FUNCTION_BLOCK FB_Euchner_MBM
VAR_INPUT
	stHwIn: ST_Euchner_MBM_HW_IN;
	bReset: BOOL;
END_VAR
VAR_OUTPUT
	stHwOut: ST_Euchner_MBM_HW_OUT;
	bError: BOOL;
	stErrorText: ST_Text;
END_VAR
VAR
	stIn: ST_Euchner_MBM_IN;
	stOut: ST_Euchner_MBM_Out;
	tonReset: ton;
END_VAR

M_Mapping();
M_Supervision();

tonReset.IN := bReset;
tonReset.PT := T#150MS;
tonReset();
IF tonReset.Q THEN
	bReset := FALSE;
END_IF
stOut.bBM_ACK_G := bReset;

METHOD PRIVATE M_Error : BOOL
VAR_INPUT
	stError: ST_Text;
END_VAR
bError	:=TRUE;
stErrorText	:= stError;
END_METHOD

METHOD PRIVATE M_Mapping : BOOL
//mapping in
stIn.bBM_D_RUN := stHwIn.nByte0.0;
stIn.bBM_E_ML1 := stHwIn.nByte0.1;
stIn.bBM_E_ML2 := stHwIn.nByte0.2;
stIn.bBM_E_SYS := stHwIn.nByte0.3;
stIn.bBM_E_G := stHwIn.nByte0.4;

//mapping in
stHwOut.nByte0.0 := stOut.bBM_ACK_G;
END_METHOD

METHOD M_Reset : BOOL
bReset	:= TRUE;
bError	:= FALSE;
MEMSET(ADR(stErrorText), 0, SiZEOF(stErrorText));
END_METHOD

METHOD PRIVATE M_Supervision : BOOL
IF stIn.bBM_E_ML1 THEN
	M_Error(F_CreateDynTextDefault("Fehler Modul MBM Starng 1")); 	
ELSIF stIn.bBM_E_ML1 THEN
	M_Error(F_CreateDynTextDefault("Fehler Modul MBM Starng 1"));	
ELSIF stIn.bBM_E_G THEN
	M_Error(F_CreateDynTextDefault("Modul MBM Allgemein"));	
ELSIF stIn.bBM_E_SYS THEN
	M_Error(F_CreateDynTextDefault("Fehler Gesamtsystem"));
END_IF
END_METHOD

END_FUNCTION_BLOCK

(* stored: Version 1.1.0.1, ProductVersion 3.1.4024.12
   POU FB_Euchner_MBM: Id {454bc480-5abf-482e-879d-5005b27308c6}, SpecialFunc None
   Method M_Error: Id {f1921ebe-4704-4a35-a03a-8bf4df5b7517}
   Method M_Mapping: Id {d872bef3-b263-479d-a742-1009d3f3c85c}
   Method M_Reset: Id {8eaf9f2b-a058-4afe-8a85-01e309ea6655}
   Method M_Supervision: Id {a4000f4a-8800-48ba-a97d-98e4ecf8db56} *)
